// TIA Portal V20 export
// export: Created 2025-12-01T14:57:02.266366Z, ExportSetting None, DisplayName Totally Integrated Automation Portal, DisplayVersion V20 Update 3, DisplayName TIA Portal Openness, DisplayVersion V20 Update 3, DisplayName TIA Portal Version Control Interface, DisplayVersion V20 Update 3, DisplayName STEP 7 Professional, DisplayVersion V20 Update 3, DisplayName STEP 7 Safety, DisplayVersion V20 Update 2, DisplayName WinCC Basic/Comfort/Advanced, DisplayVersion V20 Update 3, DisplayName WinCC Professional, DisplayVersion V20 Update 3, DisplayName WinCC Unified, DisplayVersion V20 Update 3
FUNCTION "FC420_TL_ZPA_Tarjeta_CB" : Void   // FC420, LAD
{ S7_Optimized_Access := 'FALSE' }
AUTHOR : TLigero
NAME : 20160208
VERSION : 3.3
// stored: AutoNumber false, SetENOAutomatically false
   VAR_INPUT
      Mesa : UInt;
      En_Tension : Bool;
      PhsMx : Bool;
      Avance_Tx : Bool;
      Termico_Tx : Bool;
      Simul_Mx : Bool;
      AVTF_MAnt_Mx : Bool;
      PTF_Mx_MSig : Bool;
      NXT_Avance : Bool;
      V_Paro : UDInt;   // tiempo que avanza el transportador sin aviso hasta que se para (ms)
      V_TOut_Tx_Mx : UDInt;
      V_CNT_pHsMx : UDInt;
      V_Cara_Delantera : UDInt;   // valor separación entre caras delanteras (ms)
      V_Salida : UDInt;   // hueco mínimo entre cajas (ms)
      V_Gap : UDInt;   // espacio que se deja antes de iniciar un simultaneo
   END_VAR
   VAR_OUTPUT
      PTF_MAnt_Mx : Bool;
      AVTF_Mx_MSig : Bool;
      NXT_Descarga_Act : Bool;
   END_VAR
   VAR_IN_OUT
      Mem_CNT_Salida : Bool;
      Mem_CNT_Tmp_Paro_Tx : Bool;
      Maux_FP_Marcha : Bool;
      Maux_FN_PHS : Bool;
      MAux_Descarga_activa : Bool;
      Maux_permiso_paso : Bool;
      Maux_Tok : Bool;
      Maux_flanco : Bool;
   END_VAR
   VAR_TEMP
      OK_Avance : Bool;
      cara_delantera_OK : Bool;
      fp_Marcha : Bool;
      fn_phs_tx : Bool;
      fp_phs_tx : Bool;
      Mem_CNT_Centrado : Bool;
      Mem_CNT_Gap : Bool;
      Error_atasco : Bool;
      TEMP_NXT_AVTF : Bool;
      Reset_delantera : Bool;
      OK_tension : Bool;
   END_VAR
   VAR_TEMP   // added for the SCL form of the ladder/FBD networks
      _w1 : Bool;
   END_VAR
BEGIN

REGION Network 1: Marca General Error
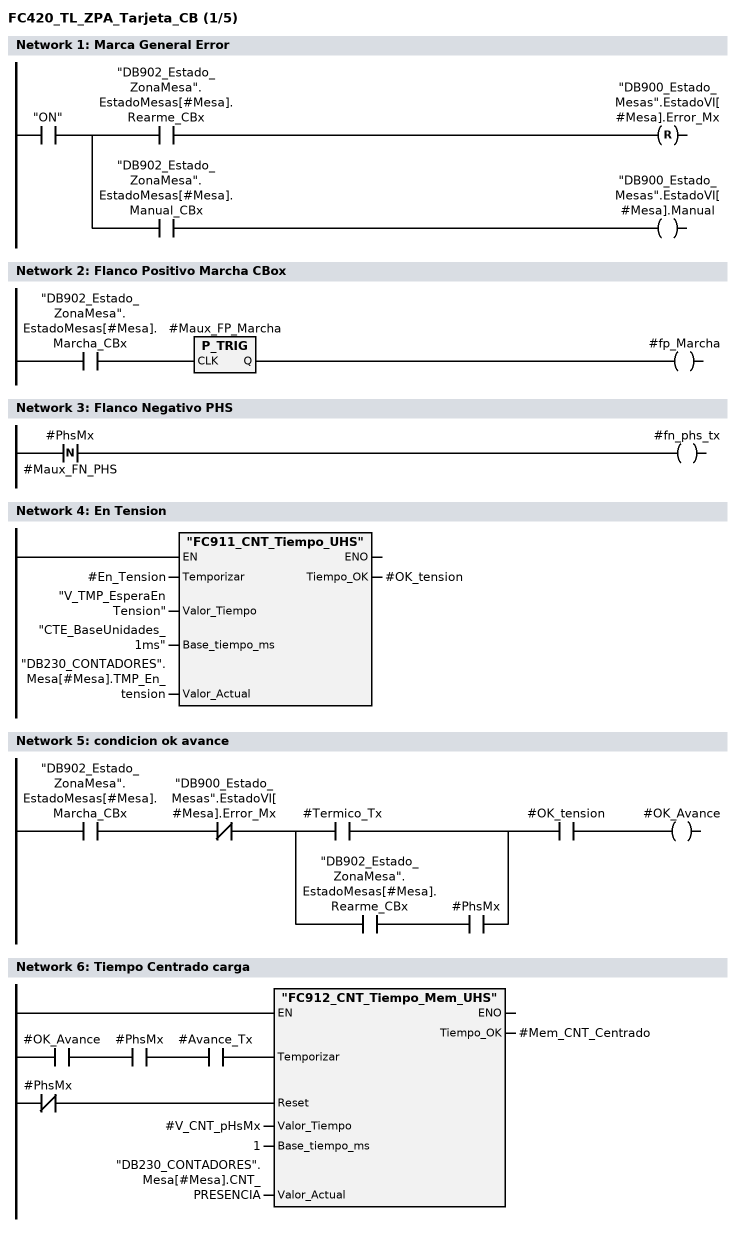
   RUNG wire#powerrail
      Contact( "ON" )
      wire#w1
      Contact( "DB902_Estado_ZonaMesa".EstadoMesas[#Mesa].Rearme_CBx )
      R_Coil( "DB900_Estado_Mesas".EstadoVI[#Mesa].Error_Mx )
   END_RUNG
   RUNG wire#w1
      Contact( "DB902_Estado_ZonaMesa".EstadoMesas[#Mesa].Manual_CBx )
      Coil( "DB900_Estado_Mesas".EstadoVI[#Mesa].Manual )
   END_RUNG
   // the same network as SCL:
   IF "ON" AND "DB902_Estado_ZonaMesa".EstadoMesas[#Mesa].Rearme_CBx THEN
       "DB900_Estado_Mesas".EstadoVI[#Mesa].Error_Mx := FALSE;
   END_IF;
   "DB900_Estado_Mesas".EstadoVI[#Mesa].Manual := "ON" AND "DB902_Estado_ZonaMesa".EstadoMesas[#Mesa].Manual_CBx;
END_REGION

REGION Network 2: Flanco Positivo Marcha CBox
   RUNG wire#powerrail
      Contact( "DB902_Estado_ZonaMesa".EstadoMesas[#Mesa].Marcha_CBx )
      P_Trig( #Maux_FP_Marcha )
      Coil( #fp_Marcha )
   END_RUNG
   // the same network as SCL:
   #_w1 := "DB902_Estado_ZonaMesa".EstadoMesas[#Mesa].Marcha_CBx AND NOT #Maux_FP_Marcha;   // rising edge
   #Maux_FP_Marcha := "DB902_Estado_ZonaMesa".EstadoMesas[#Mesa].Marcha_CBx;
   #fp_Marcha := #_w1;
END_REGION

REGION Network 3: Flanco Negativo PHS
   RUNG wire#powerrail
      N_Contact(operand := #PhsMx, bit := #Maux_FN_PHS)
      Coil( #fn_phs_tx )
   END_RUNG
   // the same network as SCL:
   #_w1 := NOT #PhsMx AND #Maux_FN_PHS;   // falling edge of #PhsMx
   #Maux_FN_PHS := #PhsMx;
   #fn_phs_tx := #_w1;
END_REGION

REGION Network 4: En Tension
   RUNG wire#powerrail
      "FC911_CNT_Tiempo_UHS"(Temporizar := #En_Tension, Valor_Tiempo := "V_TMP_EsperaEnTension", Base_tiempo_ms := "CTE_BaseUnidades_1ms", Valor_Actual := "DB230_CONTADORES".Mesa[#Mesa].TMP_En_tension, Tiempo_OK => #OK_tension)
   END_RUNG
   // the same network as SCL:
   "FC911_CNT_Tiempo_UHS"(Temporizar := #En_Tension,
                          Valor_Tiempo := "V_TMP_EsperaEnTension",
                          Base_tiempo_ms := "CTE_BaseUnidades_1ms",
                          Valor_Actual := "DB230_CONTADORES".Mesa[#Mesa].TMP_En_tension,
                          Tiempo_OK => #OK_tension);
END_REGION

REGION Network 5: condicion ok avance
   RUNG wire#powerrail
      Contact( "DB902_Estado_ZonaMesa".EstadoMesas[#Mesa].Marcha_CBx )
      I_Contact( "DB900_Estado_Mesas".EstadoVI[#Mesa].Error_Mx )
      wire#w1
      Contact( #Termico_Tx )
      wire#w2
      Contact( #OK_tension )
      Coil( #OK_Avance )
   END_RUNG
   RUNG wire#w1
      Contact( "DB902_Estado_ZonaMesa".EstadoMesas[#Mesa].Rearme_CBx )
      Contact( #PhsMx )
   END_RUNG wire#w2
   // the same network as SCL:
   #OK_Avance := "DB902_Estado_ZonaMesa".EstadoMesas[#Mesa].Marcha_CBx AND NOT "DB900_Estado_Mesas".EstadoVI[#Mesa].Error_Mx AND (#Termico_Tx OR ("DB902_Estado_ZonaMesa".EstadoMesas[#Mesa].Rearme_CBx AND #PhsMx)) AND #OK_tension;
END_REGION

REGION Network 6: Tiempo Centrado carga
   RUNG wire#powerrail
      "FC912_CNT_Tiempo_Mem_UHS"(Temporizar := wire#w1, Reset := wire#w2, Valor_Tiempo := #V_CNT_pHsMx, Base_tiempo_ms := 1, Valor_Actual := "DB230_CONTADORES".Mesa[#Mesa].CNT_PRESENCIA, Tiempo_OK => #Mem_CNT_Centrado)
   END_RUNG
   RUNG wire#powerrail
      Contact( #OK_Avance )
      Contact( #PhsMx )
      Contact( #Avance_Tx )
   END_RUNG wire#w1
   RUNG wire#powerrail
      I_Contact( #PhsMx )
   END_RUNG wire#w2
   // the same network as SCL:
   "FC912_CNT_Tiempo_Mem_UHS"(Temporizar := #OK_Avance AND #PhsMx AND #Avance_Tx,
                           Reset := NOT #PhsMx,
                           Valor_Tiempo := #V_CNT_pHsMx,
                           Base_tiempo_ms := 1,
                           Valor_Actual := "DB230_CONTADORES".Mesa[#Mesa].CNT_PRESENCIA,
                           Tiempo_OK => #Mem_CNT_Centrado);
END_REGION

REGION Network 7: contador tiempo de gap
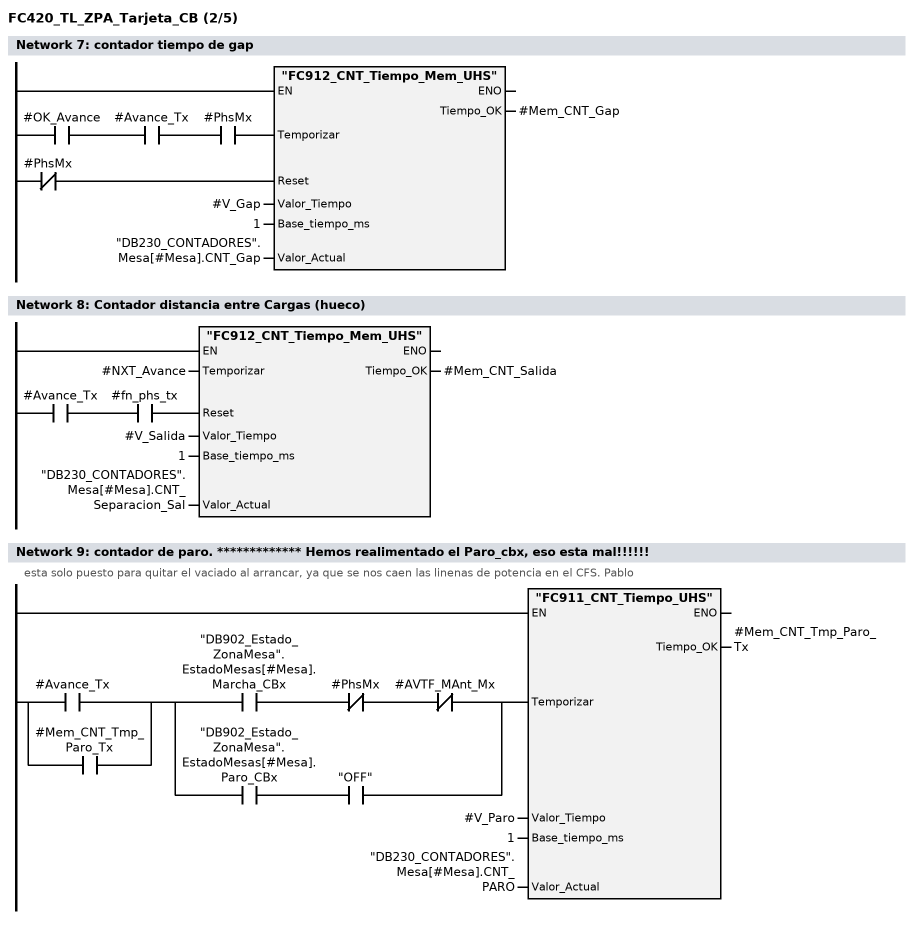
   RUNG wire#powerrail
      "FC912_CNT_Tiempo_Mem_UHS"(Temporizar := wire#w1, Reset := wire#w2, Valor_Tiempo := #V_Gap, Base_tiempo_ms := 1, Valor_Actual := "DB230_CONTADORES".Mesa[#Mesa].CNT_Gap, Tiempo_OK => #Mem_CNT_Gap)
   END_RUNG
   RUNG wire#powerrail
      Contact( #OK_Avance )
      Contact( #Avance_Tx )
      Contact( #PhsMx )
   END_RUNG wire#w1
   RUNG wire#powerrail
      I_Contact( #PhsMx )
   END_RUNG wire#w2
   // the same network as SCL:
   "FC912_CNT_Tiempo_Mem_UHS"(Temporizar := #OK_Avance AND #Avance_Tx AND #PhsMx,
                           Reset := NOT #PhsMx,
                           Valor_Tiempo := #V_Gap,
                           Base_tiempo_ms := 1,
                           Valor_Actual := "DB230_CONTADORES".Mesa[#Mesa].CNT_Gap,
                           Tiempo_OK => #Mem_CNT_Gap);
END_REGION

REGION Network 8: Contador distancia entre Cargas (hueco)
   RUNG wire#powerrail
      "FC912_CNT_Tiempo_Mem_UHS"(Reset := wire#w1, Temporizar := #NXT_Avance, Valor_Tiempo := #V_Salida, Base_tiempo_ms := 1, Valor_Actual := "DB230_CONTADORES".Mesa[#Mesa].CNT_Separacion_Sal, Tiempo_OK => #Mem_CNT_Salida)
   END_RUNG
   RUNG wire#powerrail
      Contact( #Avance_Tx )
      Contact( #fn_phs_tx )
   END_RUNG wire#w1
   // the same network as SCL:
   "FC912_CNT_Tiempo_Mem_UHS"(Temporizar := #NXT_Avance,
                           Reset := #Avance_Tx AND #fn_phs_tx,
                           Valor_Tiempo := #V_Salida,
                           Base_tiempo_ms := 1,
                           Valor_Actual := "DB230_CONTADORES".Mesa[#Mesa].CNT_Separacion_Sal,
                           Tiempo_OK => #Mem_CNT_Salida);
END_REGION

REGION Network 9: contador de paro. ************* Hemos realimentado el Paro_cbx, eso esta mal!!!!!!
   // esta solo puesto para quitar el vaciado al arrancar, ya que se nos caen las linenas de potencia en el CFS. Pablo
   RUNG wire#powerrail
      "FC911_CNT_Tiempo_UHS"(Temporizar := wire#w2, Valor_Tiempo := #V_Paro, Base_tiempo_ms := 1, Valor_Actual := "DB230_CONTADORES".Mesa[#Mesa].CNT_PARO, Tiempo_OK => #Mem_CNT_Tmp_Paro_Tx)
   END_RUNG
   RUNG wire#powerrail
      Contact( #Avance_Tx )
      wire#w1
      Contact( "DB902_Estado_ZonaMesa".EstadoMesas[#Mesa].Marcha_CBx )
      I_Contact( #PhsMx )
      I_Contact( #AVTF_MAnt_Mx )
   END_RUNG wire#w2
   RUNG wire#powerrail
      Contact( #Mem_CNT_Tmp_Paro_Tx )
   END_RUNG wire#w1
   RUNG wire#w1
      Contact( "DB902_Estado_ZonaMesa".EstadoMesas[#Mesa].Paro_CBx )
      Contact( "OFF" )
   END_RUNG wire#w2
   // the same network as SCL:
   "FC911_CNT_Tiempo_UHS"(Temporizar := (#Avance_Tx OR #Mem_CNT_Tmp_Paro_Tx) AND (("DB902_Estado_ZonaMesa".EstadoMesas[#Mesa].Marcha_CBx AND NOT #PhsMx AND NOT #AVTF_MAnt_Mx) OR ("DB902_Estado_ZonaMesa".EstadoMesas[#Mesa].Paro_CBx AND "OFF")),
                          Valor_Tiempo := #V_Paro,
                          Base_tiempo_ms := 1,
                          Valor_Actual := "DB230_CONTADORES".Mesa[#Mesa].CNT_PARO,
                          Tiempo_OK => #Mem_CNT_Tmp_Paro_Tx);
END_REGION

REGION Network 10: avance 13. QUITAMOS EL VACIADO PORQUE NOS SALTA LA FUENTE. SOLO EN CFS!!!!!!!!
   // ESTE SEGMENTO ESTA MAL!!! NNO DEBE ESTAR EL OFF EN EL FP_MARCHA. PABLO
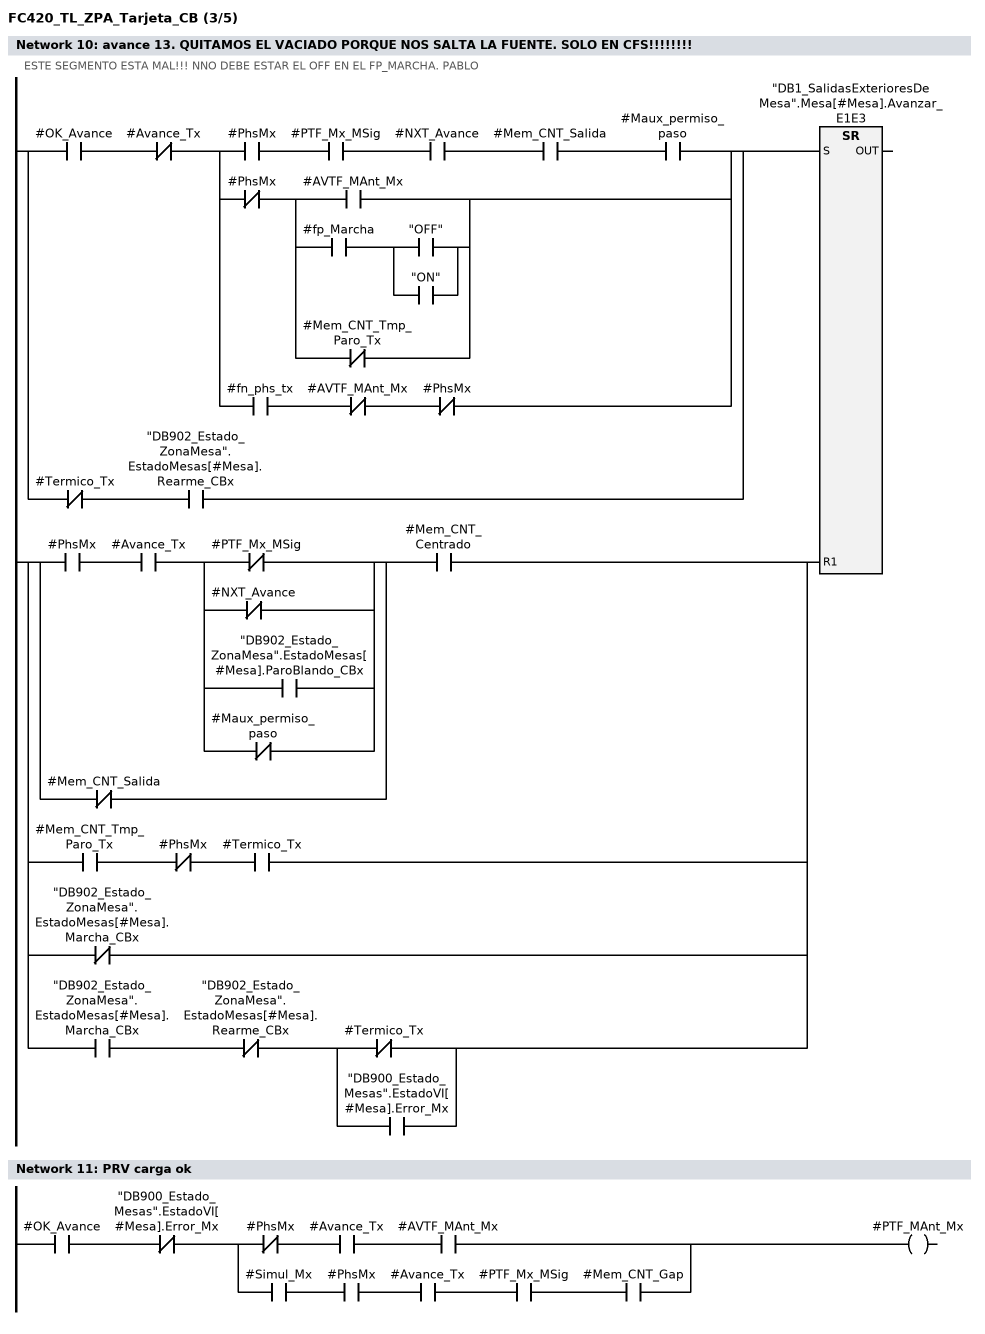
   RUNG wire#powerrail
      Contact( #OK_Avance )
      I_Contact( #Avance_Tx )
      wire#w1
      Contact( #PhsMx )
      Contact( #PTF_Mx_MSig )
      Contact( #NXT_Avance )
      Contact( #Mem_CNT_Salida )
      Contact( #Maux_permiso_paso )
      wire#w2
      S_SR(operand := "DB1_SalidasExterioresDeMesa".Mesa[#Mesa].Avanzar_E1E3, r1 := wire#w8)
   END_RUNG
   RUNG wire#w1
      I_Contact( #PhsMx )
      wire#w3
      Contact( #AVTF_MAnt_Mx )
   END_RUNG wire#w2
   RUNG wire#w3
      Contact( #fp_Marcha )
      wire#w4
      Contact( "OFF" )
   END_RUNG wire#w2
   RUNG wire#w4
      Contact( "ON" )
   END_RUNG wire#w2
   RUNG wire#w3
      I_Contact( #Mem_CNT_Tmp_Paro_Tx )
   END_RUNG wire#w2
   RUNG wire#w1
      Contact( #fn_phs_tx )
      I_Contact( #AVTF_MAnt_Mx )
      I_Contact( #PhsMx )
   END_RUNG wire#w2
   RUNG wire#powerrail
      I_Contact( #Termico_Tx )
      Contact( "DB902_Estado_ZonaMesa".EstadoMesas[#Mesa].Rearme_CBx )
   END_RUNG wire#w2
   RUNG wire#powerrail
      Contact( #PhsMx )
      Contact( #Avance_Tx )
      wire#w5
      I_Contact( #PTF_Mx_MSig )
      wire#w6
      Contact( #Mem_CNT_Centrado )
   END_RUNG wire#w8
   RUNG wire#w5
      I_Contact( #NXT_Avance )
   END_RUNG wire#w6
   RUNG wire#w5
      Contact( "DB902_Estado_ZonaMesa".EstadoMesas[#Mesa].ParoBlando_CBx )
   END_RUNG wire#w6
   RUNG wire#w5
      I_Contact( #Maux_permiso_paso )
   END_RUNG wire#w6
   RUNG wire#powerrail
      I_Contact( #Mem_CNT_Salida )
   END_RUNG wire#w6
   RUNG wire#powerrail
      Contact( #Mem_CNT_Tmp_Paro_Tx )
      I_Contact( #PhsMx )
      Contact( #Termico_Tx )
   END_RUNG wire#w8
   RUNG wire#powerrail
      I_Contact( "DB902_Estado_ZonaMesa".EstadoMesas[#Mesa].Marcha_CBx )
   END_RUNG wire#w8
   RUNG wire#powerrail
      Contact( "DB902_Estado_ZonaMesa".EstadoMesas[#Mesa].Marcha_CBx )
      I_Contact( "DB902_Estado_ZonaMesa".EstadoMesas[#Mesa].Rearme_CBx )
      wire#w7
      I_Contact( #Termico_Tx )
   END_RUNG wire#w8
   RUNG wire#w7
      Contact( "DB900_Estado_Mesas".EstadoVI[#Mesa].Error_Mx )
   END_RUNG wire#w8
   // the same network as SCL:
   #_w1 := (((#PhsMx AND #Avance_Tx AND (NOT #PTF_Mx_MSig OR NOT #NXT_Avance OR "DB902_Estado_ZonaMesa".EstadoMesas[#Mesa].ParoBlando_CBx OR NOT #Maux_permiso_paso)) OR NOT #Mem_CNT_Salida) AND #Mem_CNT_Centrado) OR (#Mem_CNT_Tmp_Paro_Tx AND NOT #PhsMx AND #Termico_Tx) OR NOT "DB902_Estado_ZonaMesa".EstadoMesas[#Mesa].Marcha_CBx OR ("DB902_Estado_ZonaMesa".EstadoMesas[#Mesa].Marcha_CBx AND NOT "DB902_Estado_ZonaMesa".EstadoMesas[#Mesa].Rearme_CBx AND (NOT #Termico_Tx OR "DB900_Estado_Mesas".EstadoVI[#Mesa].Error_Mx));
   IF (#OK_Avance AND NOT #Avance_Tx AND ((#PhsMx AND #PTF_Mx_MSig AND #NXT_Avance AND #Mem_CNT_Salida AND #Maux_permiso_paso) OR (NOT #PhsMx AND (#AVTF_MAnt_Mx OR (#fp_Marcha AND ("OFF" OR "ON")) OR NOT #Mem_CNT_Tmp_Paro_Tx)) OR (#fn_phs_tx AND NOT #AVTF_MAnt_Mx AND NOT #PhsMx))) OR (NOT #Termico_Tx AND "DB902_Estado_ZonaMesa".EstadoMesas[#Mesa].Rearme_CBx) THEN
       "DB1_SalidasExterioresDeMesa".Mesa[#Mesa].Avanzar_E1E3 := TRUE;   // SR flip-flop
   END_IF;
   IF #_w1 THEN "DB1_SalidasExterioresDeMesa".Mesa[#Mesa].Avanzar_E1E3 := FALSE; END_IF;
END_REGION

REGION Network 11: PRV carga ok
   RUNG wire#powerrail
      Contact( #OK_Avance )
      I_Contact( "DB900_Estado_Mesas".EstadoVI[#Mesa].Error_Mx )
      wire#w1
      I_Contact( #PhsMx )
      Contact( #Avance_Tx )
      Contact( #AVTF_MAnt_Mx )
      wire#w2
      Coil( #PTF_MAnt_Mx )
   END_RUNG
   RUNG wire#w1
      Contact( #Simul_Mx )
      Contact( #PhsMx )
      Contact( #Avance_Tx )
      Contact( #PTF_Mx_MSig )
      Contact( #Mem_CNT_Gap )
   END_RUNG wire#w2
   // the same network as SCL:
   #PTF_MAnt_Mx := #OK_Avance AND NOT "DB900_Estado_Mesas".EstadoVI[#Mesa].Error_Mx AND ((NOT #PhsMx AND #Avance_Tx AND #AVTF_MAnt_Mx) OR (#Simul_Mx AND #PhsMx AND #Avance_Tx AND #PTF_Mx_MSig AND #Mem_CNT_Gap));
END_REGION

REGION Network 12: NXT AVTF
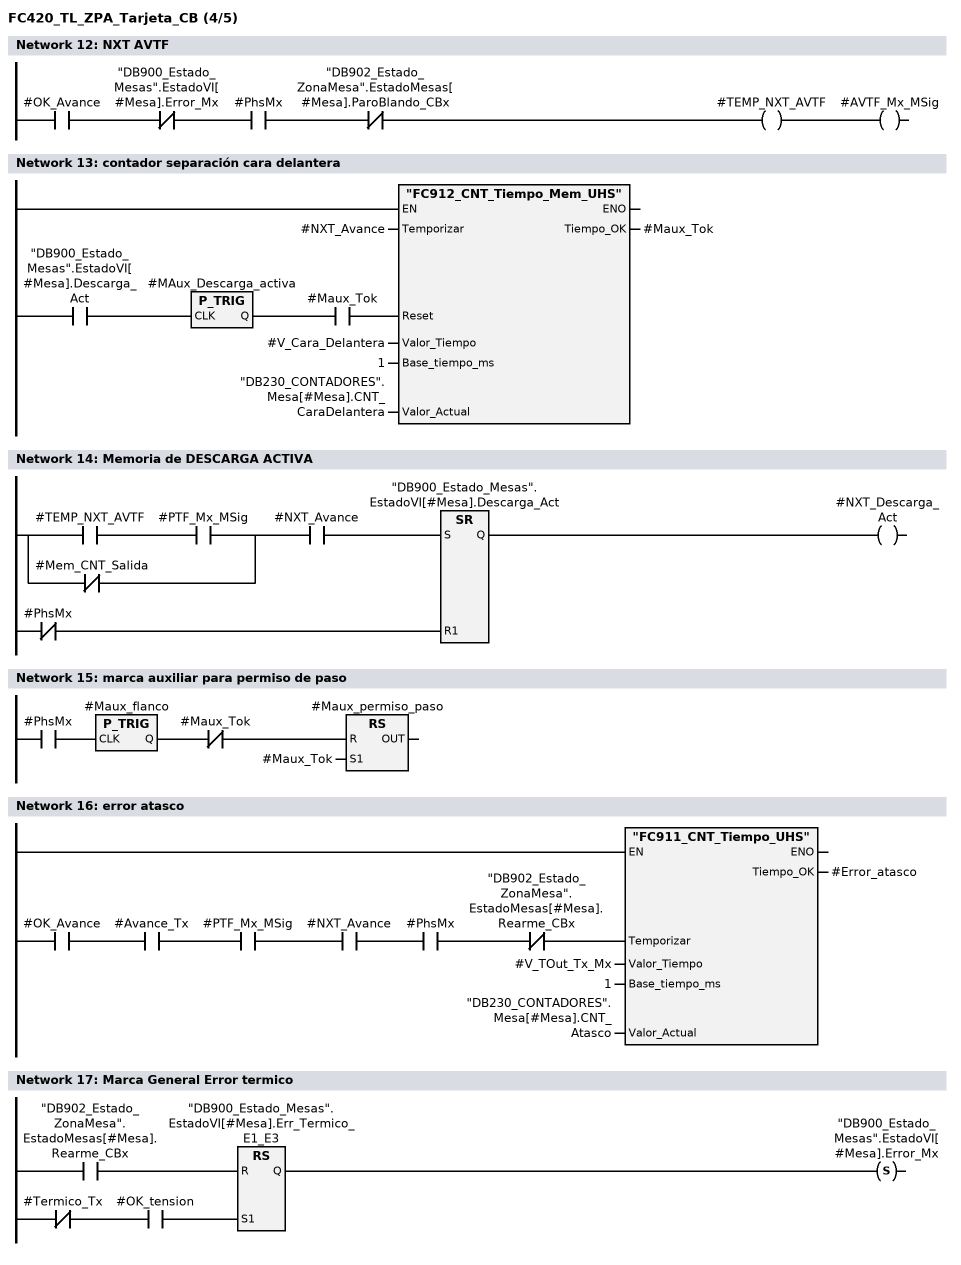
   RUNG wire#powerrail
      Contact( #OK_Avance )
      I_Contact( "DB900_Estado_Mesas".EstadoVI[#Mesa].Error_Mx )
      Contact( #PhsMx )
      I_Contact( "DB902_Estado_ZonaMesa".EstadoMesas[#Mesa].ParoBlando_CBx )
      Coil( #TEMP_NXT_AVTF )
      Coil( #AVTF_Mx_MSig )
   END_RUNG
   // the same network as SCL:
   #TEMP_NXT_AVTF := #OK_Avance AND NOT "DB900_Estado_Mesas".EstadoVI[#Mesa].Error_Mx AND #PhsMx AND NOT "DB902_Estado_ZonaMesa".EstadoMesas[#Mesa].ParoBlando_CBx;
   #AVTF_Mx_MSig := #TEMP_NXT_AVTF;
END_REGION

REGION Network 13: contador separación cara delantera
   RUNG wire#powerrail
      "FC912_CNT_Tiempo_Mem_UHS"(Reset := wire#w1, Temporizar := #NXT_Avance, Valor_Tiempo := #V_Cara_Delantera, Base_tiempo_ms := 1, Valor_Actual := "DB230_CONTADORES".Mesa[#Mesa].CNT_CaraDelantera, Tiempo_OK => #Maux_Tok)
   END_RUNG
   RUNG wire#powerrail
      Contact( "DB900_Estado_Mesas".EstadoVI[#Mesa].Descarga_Act )
      P_Trig( #MAux_Descarga_activa )
      Contact( #Maux_Tok )
   END_RUNG wire#w1
   // the same network as SCL:
   #_w1 := "DB900_Estado_Mesas".EstadoVI[#Mesa].Descarga_Act AND NOT #MAux_Descarga_activa;   // rising edge
   #MAux_Descarga_activa := "DB900_Estado_Mesas".EstadoVI[#Mesa].Descarga_Act;
   "FC912_CNT_Tiempo_Mem_UHS"(Temporizar := #NXT_Avance,
                           Reset := #_w1 AND #Maux_Tok,
                           Valor_Tiempo := #V_Cara_Delantera,
                           Base_tiempo_ms := 1,
                           Valor_Actual := "DB230_CONTADORES".Mesa[#Mesa].CNT_CaraDelantera,
                           Tiempo_OK => #Maux_Tok);
END_REGION

REGION Network 14: Memoria de DESCARGA ACTIVA
   RUNG wire#powerrail
      Contact( #TEMP_NXT_AVTF )
      Contact( #PTF_Mx_MSig )
      wire#w1
      Contact( #NXT_Avance )
      S_SR(operand := "DB900_Estado_Mesas".EstadoVI[#Mesa].Descarga_Act, r1 := wire#w2)
      Coil( #NXT_Descarga_Act )
   END_RUNG
   RUNG wire#powerrail
      I_Contact( #Mem_CNT_Salida )
   END_RUNG wire#w1
   RUNG wire#powerrail
      I_Contact( #PhsMx )
   END_RUNG wire#w2
   // the same network as SCL:
   IF ((#TEMP_NXT_AVTF AND #PTF_Mx_MSig) OR NOT #Mem_CNT_Salida) AND #NXT_Avance THEN
       "DB900_Estado_Mesas".EstadoVI[#Mesa].Descarga_Act := TRUE;   // SR flip-flop
   END_IF;
   IF NOT #PhsMx THEN "DB900_Estado_Mesas".EstadoVI[#Mesa].Descarga_Act := FALSE; END_IF;
   #NXT_Descarga_Act := "DB900_Estado_Mesas".EstadoVI[#Mesa].Descarga_Act;
END_REGION

REGION Network 15: marca auxiliar para permiso de paso
   RUNG wire#powerrail
      Contact( #PhsMx )
      P_Trig( #Maux_flanco )
      I_Contact( #Maux_Tok )
      S_RS(operand := #Maux_permiso_paso, s1 := #Maux_Tok)
   END_RUNG
   // the same network as SCL:
   #_w1 := #PhsMx AND NOT #Maux_flanco;   // rising edge
   #Maux_flanco := #PhsMx;
   IF #_w1 AND NOT #Maux_Tok THEN
       #Maux_permiso_paso := FALSE;   // RS flip-flop
   END_IF;
   IF #Maux_Tok THEN #Maux_permiso_paso := TRUE; END_IF;
END_REGION

REGION Network 16: error atasco
   RUNG wire#powerrail
      "FC911_CNT_Tiempo_UHS"(Temporizar := wire#w1, Valor_Tiempo := #V_TOut_Tx_Mx, Base_tiempo_ms := 1, Valor_Actual := "DB230_CONTADORES".Mesa[#Mesa].CNT_Atasco, Tiempo_OK => #Error_atasco)
   END_RUNG
   RUNG wire#powerrail
      Contact( #OK_Avance )
      Contact( #Avance_Tx )
      Contact( #PTF_Mx_MSig )
      Contact( #NXT_Avance )
      Contact( #PhsMx )
      I_Contact( "DB902_Estado_ZonaMesa".EstadoMesas[#Mesa].Rearme_CBx )
   END_RUNG wire#w1
   // the same network as SCL:
   "FC911_CNT_Tiempo_UHS"(Temporizar := #OK_Avance AND #Avance_Tx AND #PTF_Mx_MSig AND #NXT_Avance AND #PhsMx AND NOT "DB902_Estado_ZonaMesa".EstadoMesas[#Mesa].Rearme_CBx,
                          Valor_Tiempo := #V_TOut_Tx_Mx,
                          Base_tiempo_ms := 1,
                          Valor_Actual := "DB230_CONTADORES".Mesa[#Mesa].CNT_Atasco,
                          Tiempo_OK => #Error_atasco);
END_REGION

REGION Network 17: Marca General Error termico
   RUNG wire#powerrail
      Contact( "DB902_Estado_ZonaMesa".EstadoMesas[#Mesa].Rearme_CBx )
      S_RS(operand := "DB900_Estado_Mesas".EstadoVI[#Mesa].Err_Termico_E1_E3, s1 := wire#w1)
      S_Coil( "DB900_Estado_Mesas".EstadoVI[#Mesa].Error_Mx )
   END_RUNG
   RUNG wire#powerrail
      I_Contact( #Termico_Tx )
      Contact( #OK_tension )
   END_RUNG wire#w1
   // the same network as SCL:
   IF "DB902_Estado_ZonaMesa".EstadoMesas[#Mesa].Rearme_CBx THEN
       "DB900_Estado_Mesas".EstadoVI[#Mesa].Err_Termico_E1_E3 := FALSE;   // RS flip-flop
   END_IF;
   IF NOT #Termico_Tx AND #OK_tension THEN
       "DB900_Estado_Mesas".EstadoVI[#Mesa].Err_Termico_E1_E3 := TRUE;
   END_IF;
   IF "DB900_Estado_Mesas".EstadoVI[#Mesa].Err_Termico_E1_E3 THEN
       "DB900_Estado_Mesas".EstadoVI[#Mesa].Error_Mx := TRUE;
   END_IF;
END_REGION

REGION Network 18: Marca General Error tout avance
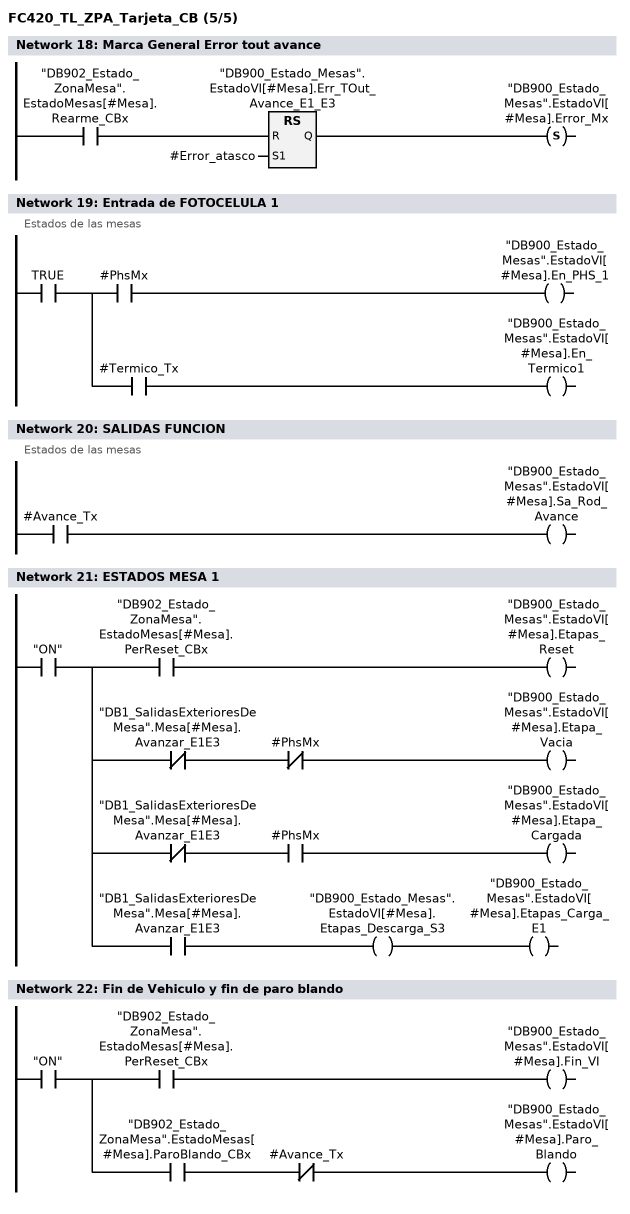
   RUNG wire#powerrail
      Contact( "DB902_Estado_ZonaMesa".EstadoMesas[#Mesa].Rearme_CBx )
      S_RS(operand := "DB900_Estado_Mesas".EstadoVI[#Mesa].Err_TOut_Avance_E1_E3, s1 := #Error_atasco)
      S_Coil( "DB900_Estado_Mesas".EstadoVI[#Mesa].Error_Mx )
   END_RUNG
   // the same network as SCL:
   IF "DB902_Estado_ZonaMesa".EstadoMesas[#Mesa].Rearme_CBx THEN
       "DB900_Estado_Mesas".EstadoVI[#Mesa].Err_TOut_Avance_E1_E3 := FALSE;   // RS flip-flop
   END_IF;
   IF #Error_atasco THEN "DB900_Estado_Mesas".EstadoVI[#Mesa].Err_TOut_Avance_E1_E3 := TRUE; END_IF;
   IF "DB900_Estado_Mesas".EstadoVI[#Mesa].Err_TOut_Avance_E1_E3 THEN
       "DB900_Estado_Mesas".EstadoVI[#Mesa].Error_Mx := TRUE;
   END_IF;
END_REGION

REGION Network 19: Entrada de FOTOCELULA 1
   // Estados de las mesas
   RUNG wire#powerrail
      Contact( TRUE )
      wire#w1
      Contact( #PhsMx )
      Coil( "DB900_Estado_Mesas".EstadoVI[#Mesa].En_PHS_1 )
   END_RUNG
   RUNG wire#w1
      Contact( #Termico_Tx )
      Coil( "DB900_Estado_Mesas".EstadoVI[#Mesa].En_Termico1 )
   END_RUNG
   // the same network as SCL:
   "DB900_Estado_Mesas".EstadoVI[#Mesa].En_PHS_1 := TRUE AND #PhsMx;
   "DB900_Estado_Mesas".EstadoVI[#Mesa].En_Termico1 := TRUE AND #Termico_Tx;
END_REGION

REGION Network 20: SALIDAS FUNCION
   // Estados de las mesas
   RUNG wire#powerrail
      Contact( #Avance_Tx )
      Coil( "DB900_Estado_Mesas".EstadoVI[#Mesa].Sa_Rod_Avance )
   END_RUNG
   // the same network as SCL:
   "DB900_Estado_Mesas".EstadoVI[#Mesa].Sa_Rod_Avance := #Avance_Tx;
END_REGION

REGION Network 21: ESTADOS MESA 1
   RUNG wire#powerrail
      Contact( "ON" )
      wire#w1
      Contact( "DB902_Estado_ZonaMesa".EstadoMesas[#Mesa].PerReset_CBx )
      Coil( "DB900_Estado_Mesas".EstadoVI[#Mesa].Etapas_Reset )
   END_RUNG
   RUNG wire#w1
      I_Contact( "DB1_SalidasExterioresDeMesa".Mesa[#Mesa].Avanzar_E1E3 )
      I_Contact( #PhsMx )
      Coil( "DB900_Estado_Mesas".EstadoVI[#Mesa].Etapa_Vacia )
   END_RUNG
   RUNG wire#w1
      I_Contact( "DB1_SalidasExterioresDeMesa".Mesa[#Mesa].Avanzar_E1E3 )
      Contact( #PhsMx )
      Coil( "DB900_Estado_Mesas".EstadoVI[#Mesa].Etapa_Cargada )
   END_RUNG
   RUNG wire#w1
      Contact( "DB1_SalidasExterioresDeMesa".Mesa[#Mesa].Avanzar_E1E3 )
      Coil( "DB900_Estado_Mesas".EstadoVI[#Mesa].Etapas_Descarga_S3 )
      Coil( "DB900_Estado_Mesas".EstadoVI[#Mesa].Etapas_Carga_E1 )
   END_RUNG
   // the same network as SCL:
   "DB900_Estado_Mesas".EstadoVI[#Mesa].Etapas_Reset := "ON" AND "DB902_Estado_ZonaMesa".EstadoMesas[#Mesa].PerReset_CBx;
   "DB900_Estado_Mesas".EstadoVI[#Mesa].Etapa_Vacia := "ON" AND NOT "DB1_SalidasExterioresDeMesa".Mesa[#Mesa].Avanzar_E1E3 AND NOT #PhsMx;
   "DB900_Estado_Mesas".EstadoVI[#Mesa].Etapa_Cargada := "ON" AND NOT "DB1_SalidasExterioresDeMesa".Mesa[#Mesa].Avanzar_E1E3 AND #PhsMx;
   #_w1 := "ON" AND "DB1_SalidasExterioresDeMesa".Mesa[#Mesa].Avanzar_E1E3;
   "DB900_Estado_Mesas".EstadoVI[#Mesa].Etapas_Descarga_S3 := #_w1;
   "DB900_Estado_Mesas".EstadoVI[#Mesa].Etapas_Carga_E1 := #_w1;
END_REGION

REGION Network 22: Fin de Vehiculo y fin de paro blando
   RUNG wire#powerrail
      Contact( "ON" )
      wire#w1
      Contact( "DB902_Estado_ZonaMesa".EstadoMesas[#Mesa].PerReset_CBx )
      Coil( "DB900_Estado_Mesas".EstadoVI[#Mesa].Fin_VI )
   END_RUNG
   RUNG wire#w1
      Contact( "DB902_Estado_ZonaMesa".EstadoMesas[#Mesa].ParoBlando_CBx )
      I_Contact( #Avance_Tx )
      Coil( "DB900_Estado_Mesas".EstadoVI[#Mesa].Paro_Blando )
   END_RUNG
   // the same network as SCL:
   "DB900_Estado_Mesas".EstadoVI[#Mesa].Fin_VI := "ON" AND "DB902_Estado_ZonaMesa".EstadoMesas[#Mesa].PerReset_CBx;
   "DB900_Estado_Mesas".EstadoVI[#Mesa].Paro_Blando := "ON" AND "DB902_Estado_ZonaMesa".EstadoMesas[#Mesa].ParoBlando_CBx AND NOT #Avance_Tx;
END_REGION
END_FUNCTION
